{attribute 'GeneratedUsingTerminal: EL6631-0000-0016'}
{attribute addProperty BoxType "EL6631-0000-0016"}
{attribute addProperty Description "EL6631 PROFINET IO Controller"}
{attribute addProperty Physics "KK"}
{attribute addProperty Id "InfoDataAT %I*InfoData_90184F0C16"}
{attribute addProperty CRC "554310285"}
{attribute addProperty Size "16"}
TYPE EL6631_210A1A8D EXTENDS EtcSlaveTerminalBase_947E5A46 :
STRUCT
	{attribute addProperty Name "InfoData"}
	InfoData : InfoData_90184F0C;
END_STRUCT
END_TYPE

(* stored: Version 1.2.0.0, ProductVersion 3.1.4024.9
   DUT EL6631_210A1A8D: Id {030d4f07-ad09-49ab-b5f9-3316d592babc} *)
